TYPE udt_HDL_PartData :
STRUCT
PartId	:DINT; //Unique Part Id (DMC Serial Number)
State	:BOOL; //Part state 0=OK, 1=NOK
Types :	BOOL;// Part type 1=Long, 0=Short
Exists	:BOOL; //Part exist


END_STRUCT
END_TYPE

(* stored: Version 1.1.0.1, ProductVersion 3.1.4024.16
   DUT udt_HDL_PartData: Id {2b238a6e-c541-437e-9e7a-7e0d4446560d} *)
